FUNCTION fPlatformAngleTheta1 : LREAL
VAR_INPUT
	fStroke : LREAL;
	
END_VAR
VAR_OUTPUT
	fPlatformAngle : LREAL;
END_VAR
VAR
	fAngleBeta		: LREAL;
	fCylinderLength	: LREAL;
	fMinLength 		: LREAL; 
END_VAR

fMinLength := G_StablePlatformParameters.fMinLengthPlatformCylinder;

fCylinderLength := fStroke + fMinLength;

fAngleBeta := ACOS((G_StablePlatformParameters.fLengthA*G_StablePlatformParameters.fLengthA +  G_StablePlatformParameters.fLengthC*G_StablePlatformParameters.fLengthC - fCylinderLength*fCylinderLength) / (2 * G_StablePlatformParameters.fLengthA * G_StablePlatformParameters.fLengthC));

fPlatformAngle := -(fAngleBeta - G_StablePlatformParameters.fOffsetAngleRad);

END_FUNCTION

(* stored: Version 1.1.0.1, ProductVersion 3.1.4024.12
   POU fPlatformAngleTheta1: Id {38f34970-9559-42d3-b750-b6b988181f54}, SpecialFunc None *)
